// TIA Portal V19 export
TYPE "Prod_Coil_Ctrl"
// stored: Access Published
   STRUCT
      Setup_LinePreparation_Exe : Bool;
      STOP_Provino : Bool;
      ACK_Provino : Bool;
      STOP_Taglio_Fine_Ordini : Bool;
      STOP_Manca_Dati_AspoInLinea : Bool;
      STOP_Manca_Dati_AspoInCarico : Bool;
      STOP_FineTurno : Bool;
      STOP_ControlloQualita : Bool;
   END_STRUCT;
END_TYPE
